FUNCTION "_toggleBit" : Void
TITLE = Function:Toggle bit
{ S7_Optimized_Access := 'TRUE' }
AUTHOR : cyanezf
FAMILY : util
NAME : _toggleBit
VERSION : 1.0

VAR_IN_OUT
      bit : Bool;
   END_VAR


BEGIN
(*--

# Log
| version | date | author | description |
|:-------:|:----:|:------:|:------------|
| v1.0 | 2018-05-13 | cyanezf | First version |

# Dependencies
| Dependency |
|:-----------|

# Description
This function toggles `bit` inout.

#
_Use [Markdown Live Preview](https://markdownlivepreview.com/) to watch this doc._
--*)

	#bit := NOT #bit;
	ENO := true;

END_FUNCTION

